// TIA Portal project "iç mekan havalandırma" (V16)

(* hardware
DEVICE "S7-1200 station_1"  S7-1200 Station
   slot 0: "Rack_0"  S7-1200 Rack  Rack  V1.0
   slot 1: "PLC_1"  CPU 1215C DC/DC/Rly  6ES7 215-1HG40-0XB0  V4.4
   slot 2: "AQ 4x14BIT_1"  6ES7 232-4HD32-0XB0  V2.1
   slot 3: "AQ 4x14BIT_2"  6ES7 232-4HD32-0XB0  V2.1
   slot 4: "AI 4xTC_1"  SM 1231 AI4 x TC  6ES7 231-5QD32-0XB0  V2.0
*)

// ===== PLC "PLC_1"  CPU 1215C DC/DC/Rly =====

VAR_GLOBAL   // PLC tag table "Default tag table"
   "start but" AT %I0.0 : Bool;
   "stop but" AT %I0.1 : Bool;
   "düşük sıcaklık lam" AT %Q0.0 : Bool;
   "normla sıcaklık lam" AT %Q0.1 : Bool;
   "yüksek sıcaklık lam" AT %Q0.2 : Bool;
   "çokyüksek sıcaklık lam" AT %Q0.3 : Bool;
   "sistem start" AT %M10.0 : Bool;
   "TERMO CUP." AT %IW30 : Word;
   "Tag_2" AT %MW20 : Word;
   "Tag_3" AT %MW22 : Word;
   "Tag_4" AT %MD22 : Real;
   "ÖLÇÜLEN SICAKLIK DEĞERİ" AT %MD26 : Real;
   "FAN1" AT %QW96 : Int;
   "FAN2" AT %QW98 : Int;
   "FAN3" AT %QW100 : Int;
   "FAN4" AT %QW102 : Int;
   "FAN5" AT %QW112 : Int;
   "FAN6" AT %QW114 : Int;
   "çok yüksek sıklık lambası mem" AT %M10.1 : Bool;
   "Clock_Byte" AT %MB0 : Byte;
   "Clock_10Hz" AT %M0.0 : Bool;
   "Clock_5Hz" AT %M0.1 : Bool;
   "Clock_2.5Hz" AT %M0.2 : Bool;
   "Clock_2Hz" AT %M0.3 : Bool;
   "Clock_1.25Hz" AT %M0.4 : Bool;
   "Clock_1Hz" AT %M0.5 : Bool;
   "Clock_0.625Hz" AT %M0.6 : Bool;
   "Clock_0.5Hz" AT %M0.7 : Bool;
   "çok yüksek sıcaklık mem 2" AT %M10.2 : Bool;
END_VAR

ORGANIZATION_BLOCK "Main"   // OB1, LAD, ProgramCycle
TITLE = "Main Program Sweep (Cycle)"
{ S7_Optimized_Access := 'TRUE' }
VERSION : 0.1
   VAR_INPUT
      Initial_Call : Bool;   // Initial call of this OB
      Remanence : Bool;   // =True, if remanent data are available
   END_VAR
   VAR_TEMP   // added for the SCL form of the ladder/FBD networks
      _w1 : Bool;
   END_VAR
BEGIN

REGION Network 1
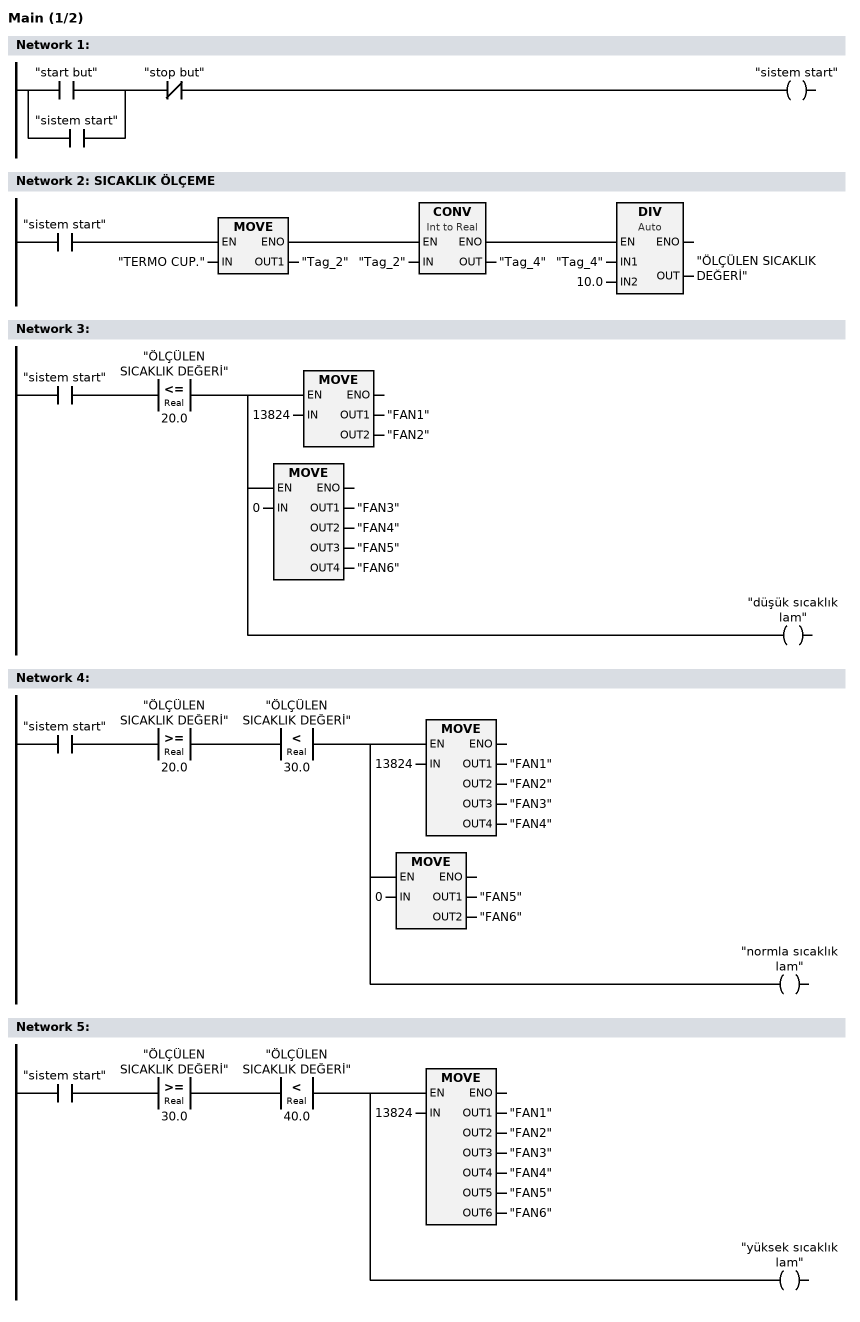
   RUNG wire#powerrail
      Contact( "start but" )
      wire#w1
      I_Contact( "stop but" )
      Coil( "sistem start" )
   END_RUNG
   RUNG wire#powerrail
      Contact( "sistem start" )
   END_RUNG wire#w1
   // the same network as SCL:
   "sistem start" := ("start but" OR "sistem start") AND NOT "stop but";
END_REGION

REGION Network 2: SICAKLIK ÖLÇEME
   RUNG wire#powerrail
      Contact( "sistem start" )
      Move(in := "TERMO CUP.", out1 => "Tag_2")
      { S7_Templates := "[SrcType := Int, DestType := Real]" } Convert(in := "Tag_2", out => "Tag_4")
      Div(in1 := "Tag_4", in2 := 10.0, out => "ÖLÇÜLEN SICAKLIK DEĞERİ")
   END_RUNG
   // the same network as SCL:
   IF "sistem start" THEN
       "Tag_2" := "TERMO CUP.";
       "Tag_4" := INT_TO_REAL("Tag_2");
       "ÖLÇÜLEN SICAKLIK DEĞERİ" := "Tag_4" / 10.0;
   END_IF;
END_REGION

REGION Network 3
   RUNG wire#powerrail
      Contact( "sistem start" )
      { S7_Templates := "SrcType := Real" } LE_Contact(in1 := "ÖLÇÜLEN SICAKLIK DEĞERİ", in2 := 20.0)
      wire#w1
      Move(in := 13824, out1 => "FAN1", out2 => "FAN2")
   END_RUNG
   RUNG wire#w1
      Move(in := 0, out1 => "FAN3", out2 => "FAN4", out3 => "FAN5", out4 => "FAN6")
   END_RUNG
   RUNG wire#w1
      Coil( "düşük sıcaklık lam" )
   END_RUNG
   // the same network as SCL:
   #_w1 := "sistem start" AND ("ÖLÇÜLEN SICAKLIK DEĞERİ" <= 20.0);
   IF #_w1 THEN
       "FAN1" := 13824;
       "FAN2" := 13824;
       "FAN3" := 0;
       "FAN4" := 0;
       "FAN5" := 0;
       "FAN6" := 0;
   END_IF;
   "düşük sıcaklık lam" := #_w1;
END_REGION

REGION Network 4
   RUNG wire#powerrail
      Contact( "sistem start" )
      { S7_Templates := "SrcType := Real" } GE_Contact(in1 := "ÖLÇÜLEN SICAKLIK DEĞERİ", in2 := 20.0)
      { S7_Templates := "SrcType := Real" } LT_Contact(in1 := "ÖLÇÜLEN SICAKLIK DEĞERİ", in2 := 30.0)
      wire#w1
      Move(in := 13824, out1 => "FAN1", out2 => "FAN2", out3 => "FAN3", out4 => "FAN4")
   END_RUNG
   RUNG wire#w1
      Move(in := 0, out1 => "FAN5", out2 => "FAN6")
   END_RUNG
   RUNG wire#w1
      Coil( "normla sıcaklık lam" )
   END_RUNG
   // the same network as SCL:
   #_w1 := "sistem start" AND ("ÖLÇÜLEN SICAKLIK DEĞERİ" >= 20.0) AND ("ÖLÇÜLEN SICAKLIK DEĞERİ" < 30.0);
   IF #_w1 THEN
       "FAN1" := 13824;
       "FAN2" := 13824;
       "FAN3" := 13824;
       "FAN4" := 13824;
       "FAN5" := 0;
       "FAN6" := 0;
   END_IF;
   "normla sıcaklık lam" := #_w1;
END_REGION

REGION Network 5
   RUNG wire#powerrail
      Contact( "sistem start" )
      { S7_Templates := "SrcType := Real" } GE_Contact(in1 := "ÖLÇÜLEN SICAKLIK DEĞERİ", in2 := 30.0)
      { S7_Templates := "SrcType := Real" } LT_Contact(in1 := "ÖLÇÜLEN SICAKLIK DEĞERİ", in2 := 40.0)
      wire#w1
      Move(in := 13824, out1 => "FAN1", out2 => "FAN2", out3 => "FAN3", out4 => "FAN4", out5 => "FAN5", out6 => "FAN6")
   END_RUNG
   RUNG wire#w1
      Coil( "yüksek sıcaklık lam" )
   END_RUNG
   // the same network as SCL:
   #_w1 := "sistem start" AND ("ÖLÇÜLEN SICAKLIK DEĞERİ" >= 30.0) AND ("ÖLÇÜLEN SICAKLIK DEĞERİ" < 40.0);
   IF #_w1 THEN
       "FAN1" := 13824;
       "FAN2" := 13824;
       "FAN3" := 13824;
       "FAN4" := 13824;
       "FAN5" := 13824;
       "FAN6" := 13824;
   END_IF;
   "yüksek sıcaklık lam" := #_w1;
END_REGION

REGION Network 6
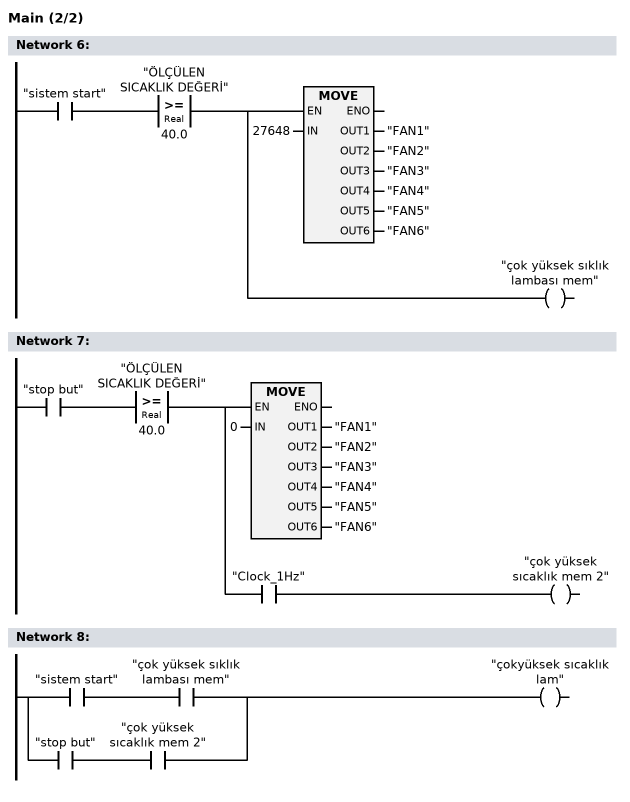
   RUNG wire#powerrail
      Contact( "sistem start" )
      { S7_Templates := "SrcType := Real" } GE_Contact(in1 := "ÖLÇÜLEN SICAKLIK DEĞERİ", in2 := 40.0)
      wire#w1
      Move(in := 27648, out1 => "FAN1", out2 => "FAN2", out3 => "FAN3", out4 => "FAN4", out5 => "FAN5", out6 => "FAN6")
   END_RUNG
   RUNG wire#w1
      Coil( "çok yüksek sıklık lambası mem" )
   END_RUNG
   // the same network as SCL:
   #_w1 := "sistem start" AND ("ÖLÇÜLEN SICAKLIK DEĞERİ" >= 40.0);
   IF #_w1 THEN
       "FAN1" := 27648;
       "FAN2" := 27648;
       "FAN3" := 27648;
       "FAN4" := 27648;
       "FAN5" := 27648;
       "FAN6" := 27648;
   END_IF;
   "çok yüksek sıklık lambası mem" := #_w1;
END_REGION

REGION Network 7
   RUNG wire#powerrail
      Contact( "stop but" )
      { S7_Templates := "SrcType := Real" } GE_Contact(in1 := "ÖLÇÜLEN SICAKLIK DEĞERİ", in2 := 40.0)
      wire#w1
      Move(in := 0, out1 => "FAN1", out2 => "FAN2", out3 => "FAN3", out4 => "FAN4", out5 => "FAN5", out6 => "FAN6")
   END_RUNG
   RUNG wire#w1
      Contact( "Clock_1Hz" )
      Coil( "çok yüksek sıcaklık mem 2" )
   END_RUNG
   // the same network as SCL:
   #_w1 := "stop but" AND ("ÖLÇÜLEN SICAKLIK DEĞERİ" >= 40.0);
   IF #_w1 THEN
       "FAN1" := 0;
       "FAN2" := 0;
       "FAN3" := 0;
       "FAN4" := 0;
       "FAN5" := 0;
       "FAN6" := 0;
   END_IF;
   "çok yüksek sıcaklık mem 2" := #_w1 AND "Clock_1Hz";
END_REGION

REGION Network 8
   RUNG wire#powerrail
      Contact( "sistem start" )
      Contact( "çok yüksek sıklık lambası mem" )
      wire#w1
      Coil( "çokyüksek sıcaklık lam" )
   END_RUNG
   RUNG wire#powerrail
      Contact( "stop but" )
      Contact( "çok yüksek sıcaklık mem 2" )
   END_RUNG wire#w1
   // the same network as SCL:
   "çokyüksek sıcaklık lam" := ("sistem start" AND "çok yüksek sıklık lambası mem") OR ("stop but" AND "çok yüksek sıcaklık mem 2");
END_REGION
END_ORGANIZATION_BLOCK